(* Logix 5000 project; controller CuteLogix vendor 1 type 14 code 216 rev 30.14; software revision 30.00 *)

TASK EventTask (event, rate 10 ms, priority 10, watchdog 500 ms) : Duh
TASK MainTask (continuous, watchdog 500 ms) : Instructions, Branching

MODULES
   Local : vendor 1 type 14 code 216 (5069 0, rev 30.14)
END_MODULES

TYPE STRING20 :
STRUCT
   LEN : DINT;
   DATA : SINT[20];
END_STRUCT
END_TYPE

VAR_GLOBAL   (* controller tags *)
   AdvancedMath : DINT[10] := ([0] := 651, [3] := 954, [6] := 6);
   ASCII : STRING[20];
   ASCII_Find : DINT;
   ASCII_Find_Result : DINT;
   ASCII_Qty : DINT;
   ASCII_Start : DINT;
   AverageControl : CONTROL := (LEN := 10);
   b_Timer : TIMER[10] := ([0].PRE := 90000, [0].ACC := 52845, [0].EN := 1, [0].TT := 1);
        [0]   // I'm a 90 Second timer
   Bits : DINT[10];
   Branching : DINT[1000] := ([0] := 82407, [1] := 11343, [2] := 76767, [3] := 20431, [4] := 93845, [5] := 88961, [6] := 95802, [7] := 76730, [8] := 78742, [9] := 28858, [10] := 24388, [11] := 98780, [12] := 74194, [13] := 88651, [14] := 97109, [15] := 70489, [16] := 21759, [17] := 12682, [18] := 51608, [19] := 51105, [20] := 34340, [21] := 67477, [22] := 9682, [23] := 52316, [24] := 60079, [25] := 87946, [26] := 25355, [27] := 61705, [28] := 23349, [29] := 32270, [30] := 4523, [31] := 20763, [32] := 39925, [33] := 47227, [34] := 25474, [35] := 90216, [36] := 63189, [37] := 19334, [38] := 13116, [39] := 58964, [40] := 74627, [41] := 92119, [42] := 81781, [43] := 93714, [44] := 35797, [45] := 72290, [46] := 23509, [47] := 2660, [48] := 45984, [49] := 72685, [50] := 48944, [51] := 54255, [52] := 57274, [53] := 86876, [54] := 25860, [55] := 34445, [56] := 55068, [57] := 196, [58] := 23518, [59] := 53104,
        [60] := 75775, [61] := 34032, [62] := 11808, [63] := 83613, [64] := 27078, [65] := 52948, [66] := 91266, [67] := 23342, [68] := 61979, [69] := 88356, [70] := 87538, [71] := 49455, [72] := 73754, [73] := 19956, [74] := 8441, [75] := 44039, [76] := 47792, [77] := 24338, [78] := 1813, [79] := 81080, [80] := 28038, [81] := 22213, [82] := 76032, [83] := 43482, [84] := 43490, [85] := 56586, [86] := 14618, [87] := 67641, [88] := 82887, [89] := 73251, [90] := 36535, [91] := 99267, [92] := 921, [93] := 34224, [94] := 81286, [95] := 89074, [96] := 74192, [97] := 35254, [98] := 70789, [99] := 94903, [100] := 90087, [101] := 75614, [102] := 74924, [103] := 66053, [104] := 67686, [105] := 14094, [106] := 50491, [107] := 19788, [108] := 36949, [109] := 46559, [110] := 33619, [111] := 72776, [112] := 43045, [113] := 66611, [114] := 49748, [115] := 23967, [116] := 66838, [117] := 33653, [118] := 92725, [119] := 32432,
        [120] := 35949, [121] := 75581, [122] := 92310, [123] := 38436, [124] := 62405, [125] := 99027, [126] := 5445, [127] := 23446, [128] := 3634, [129] := 95984, [130] := 50572, [131] := 64179, [132] := 42294, [133] := 43241, [134] := 6544, [135] := 41013, [136] := 98800, [137] := 16177, [138] := 15917, [139] := 31322, [140] := 95598, [141] := 46619, [142] := 76555, [143] := 58340, [144] := 27140, [145] := 10620, [146] := 62592, [147] := 70487, [148] := 12865, [149] := 27943, [150] := 6446, [151] := 12547, [152] := 15055, [153] := 51388, [154] := 85199, [155] := 83609, [156] := 47725, [157] := 55131, [158] := 24907, [159] := 16737, [160] := 43899, [161] := 81924, [162] := 9125, [163] := 64948, [164] := 14057, [165] := 26270, [166] := 26481, [167] := 27516, [168] := 13940, [169] := 41111, [170] := 22715, [171] := 54684, [172] := 27850, [173] := 95551, [174] := 76562, [175] := 10807, [176] := 3604, [177] := 81954, [178] := 85877, [179] := 90731,
        [180] := 50124, [181] := 84444, [182] := 93795, [183] := 58321, [184] := 83942, [185] := 55706, [186] := 21776, [187] := 72127, [188] := 98888, [189] := 98078, [190] := 46603, [191] := 5622, [192] := 2259, [193] := 25464, [194] := 68812, [195] := 39572, [196] := 82910, [197] := 30899, [198] := 41853, [199] := 18720, [200] := 32673, [201] := 51959, [202] := 85552, [203] := 56119, [204] := 37568, [205] := 65908, [206] := 29436, [207] := 79651, [208] := 34700, [209] := 32924, [210] := 83907, [211] := 40689, [212] := 52367, [213] := 8949, [214] := 33429, [215] := 68883, [216] := 57307, [217] := 85633, [218] := 56031, [219] := 3577, [220] := 79663, [221] := 84961, [222] := 38978, [223] := 80380, [224] := 69012, [225] := 39942, [226] := 80323, [227] := 51518, [228] := 32713, [229] := 15043, [230] := 11143, [231] := 84668, [232] := 62808, [233] := 99189, [234] := 72567, [235] := 21806, [236] := 89789, [237] := 79147, [238] := 40667, [239] := 99508,
        [240] := 90600, [241] := 67080, [242] := 66939, [243] := 32495, [244] := 93170, [245] := 53515, [246] := 20470, [247] := 39580, [248] := 483, [249] := 62424, [250] := 1307, [251] := 82788, [252] := 9479, [253] := 67332, [254] := 3775, [255] := 39510, [256] := 4284, [257] := 93272, [258] := 16406, [259] := 65799, [260] := 13395, [261] := 71017, [262] := 52104, [263] := 27877, [264] := 840, [265] := 28148, [266] := 57193, [267] := 76840, [268] := 15114, [269] := 73046, [270] := 48035, [271] := 68111, [272] := 12541, [273] := 80659, [274] := 7877, [275] := 15975, [276] := 56634, [277] := 47037, [278] := 15404, [279] := 7082, [280] := 97238, [281] := 3431, [282] := 79807, [283] := 43357, [284] := 57116, [285] := 78602, [286] := 23732, [287] := 6885, [288] := 94485, [289] := 44571, [290] := 96772, [291] := 35862, [292] := 88252, [293] := 11874, [294] := 63250, [295] := 96749, [296] := 34190, [297] := 12853, [298] := 29560, [299] := 61009,
        [300] := 24219, [301] := 53874, [302] := 98911, [303] := 19166, [304] := 43701, [305] := 69509, [306] := 3825, [307] := 96142, [308] := 42271, [309] := 29331, [310] := 27095, [311] := 39467, [312] := 44548, [313] := 41271, [314] := 87555, [315] := 97136, [316] := 39244, [317] := 16499, [318] := 61732, [319] := 81001, [320] := 81261, [321] := 95891, [322] := 42237, [323] := 43180, [324] := 44778, [325] := 92930, [326] := 54868, [327] := 40795, [328] := 52161, [329] := 19185, [330] := 46809, [331] := 28074, [332] := 11466, [333] := 82810, [334] := 88188, [335] := 72177, [336] := 49604, [337] := 53088, [338] := 16845, [339] := 70569, [340] := 84274, [341] := 92660, [342] := 63169, [343] := 40489, [344] := 26218, [345] := 30561, [346] := 14751, [347] := 75624, [348] := 38033, [349] := 92852, [350] := 85778, [351] := 64491, [352] := 80319, [353] := 8699, [354] := 74387, [355] := 66643, [356] := 62603, [357] := 70896, [358] := 51215, [359] := 45712,
        [360] := 55357, [361] := 77462, [362] := 64150, [363] := 15112, [364] := 85523, [365] := 32571, [366] := 68709, [367] := 30297, [368] := 99879, [369] := 99236, [370] := 14376, [371] := 42664, [372] := 53669, [373] := 22296, [374] := 32196, [375] := 17960, [376] := 42810, [377] := 28932, [378] := 99353, [379] := 54203, [380] := 52001, [381] := 4016, [382] := 41782, [383] := 26979, [384] := 19158, [385] := 41232, [386] := 97013, [387] := 55977, [388] := 62866, [389] := 30951, [390] := 77905, [391] := 86629, [392] := 59774, [393] := 197, [394] := 52381, [395] := 92029, [396] := 94556, [397] := 36193, [398] := 53622, [399] := 26385, [400] := 43506, [401] := 64525, [402] := 50552, [403] := 42062, [404] := 93734, [405] := 66267, [406] := 1973, [407] := 82396, [408] := 20210, [409] := 87, [410] := 31043, [411] := 12651, [412] := 18796, [413] := 74789, [414] := 76255, [415] := 7847, [416] := 88827, [417] := 99325, [418] := 62264, [419] := 83107,
        [420] := 54708, [421] := 81244, [422] := 3333, [423] := 82540, [424] := 76390, [425] := 976, [426] := 94348, [427] := 18663, [428] := 98314, [429] := 90843, [430] := 92080, [431] := 97486, [432] := 42367, [433] := 8830, [434] := 35849, [435] := 15548, [436] := 99329, [437] := 44884, [438] := 60276, [439] := 65875, [440] := 34626, [441] := 31589, [442] := 84178, [443] := 15627, [444] := 14886, [445] := 65838, [446] := 93540, [447] := 14359, [448] := 13136, [449] := 83951, [450] := 94714, [451] := 39093, [452] := 97112, [453] := 22873, [454] := 41442, [455] := 99078, [456] := 11004, [457] := 65685, [458] := 85926, [459] := 55000, [460] := 91532, [461] := 79264, [462] := 3410, [463] := 41917, [464] := 8700, [465] := 15683, [466] := 83367, [467] := 71772, [468] := 14428, [469] := 31148, [470] := 43290, [471] := 73920, [472] := 96383, [473] := 57141, [474] := 28794, [475] := 15145, [476] := 77125, [477] := 35399, [478] := 32019, [479] := 89297,
        [480] := 11057, [481] := 12415, [482] := 54611, [483] := 42077, [484] := 78428, [485] := 33488, [486] := 13887, [487] := 52219, [488] := 37547, [489] := 48567, [490] := 7929, [491] := 45872, [492] := 23879, [493] := 36974, [494] := 97930, [495] := 10005, [496] := 2990, [497] := 51310, [498] := 45690, [499] := 52666, [500] := 16987, [501] := 84869, [502] := 58178, [503] := 95604, [504] := 77205, [505] := 66416, [506] := 46278, [507] := 99665, [508] := 72977, [509] := 58733, [510] := 50420, [511] := 59898, [512] := 18286, [513] := 36589, [514] := 34816, [515] := 47992, [516] := 50582, [517] := 90684, [518] := 46443, [519] := 51027, [520] := 64473, [521] := 72799, [522] := 68183, [523] := 33719, [524] := 81364, [525] := 73595, [526] := 99507, [527] := 47306, [528] := 95179, [529] := 46851, [530] := 86803, [531] := 70881, [532] := 12477, [533] := 75439, [534] := 76539, [535] := 95435, [536] := 45897, [537] := 68412, [538] := 59806, [539] := 8448,
        [540] := 54361, [541] := 83177, [542] := 38861, [543] := 28242, [544] := 24846, [545] := 71585, [546] := 59255, [547] := 99852, [548] := 59975, [549] := 65189, [550] := 78689, [551] := 11674, [552] := 49631, [553] := 89733, [554] := 84628, [555] := 44306, [556] := 69954, [557] := 7239, [558] := 30285, [559] := 49616, [560] := 21695, [561] := 14771, [562] := 902, [563] := 43262, [564] := 32396, [565] := 10532, [566] := 80170, [567] := 22340, [568] := 77422, [569] := 3135, [570] := 24402, [571] := 76735, [572] := 20681, [573] := 94053, [574] := 74442, [575] := 18763, [576] := 9089, [577] := 88936, [578] := 46733, [579] := 47489, [580] := 36126, [581] := 46401, [582] := 56328, [583] := 96948, [584] := 6036, [585] := 61754, [586] := 98282, [587] := 41889, [588] := 9356, [589] := 80694, [590] := 51720, [591] := 56107, [592] := 99379, [593] := 42488, [594] := 63660, [595] := 79873, [596] := 46147, [597] := 44287, [598] := 62154, [599] := 55518,
        [600] := 7753, [601] := 47609, [602] := 31410, [603] := 49961, [604] := 52145, [605] := 16507, [606] := 34414, [607] := 81979, [608] := 23958, [609] := 86010, [610] := 94833, [611] := 89494, [612] := 82851, [613] := 94123, [614] := 60739, [615] := 38788, [616] := 88402, [617] := 62854, [618] := 49018, [619] := 53666, [620] := 9949, [621] := 25600, [622] := 11619, [623] := 73987, [624] := 94764, [625] := 51443, [626] := 42099, [627] := 43731, [628] := 17824, [629] := 20355, [630] := 25854, [631] := 69789, [632] := 6342, [633] := 67396, [634] := 79990, [635] := 20527, [636] := 18543, [637] := 40174, [638] := 10905, [639] := 15107, [640] := 13163, [641] := 12315, [642] := 79884, [643] := 18443, [644] := 64372, [645] := 31725, [646] := 31353, [647] := 31436, [648] := 91466, [649] := 57461, [650] := 73514, [651] := 7803, [652] := 83871, [653] := 95183, [654] := 29573, [655] := 19778, [656] := 58366, [657] := 60531, [658] := 76491, [659] := 47189,
        [660] := 17277, [661] := 81754, [662] := 59413, [663] := 83709, [664] := 10893, [665] := 45396, [666] := 98708, [667] := 59876, [668] := 13826, [669] := 67604, [670] := 55566, [671] := 64210, [672] := 14166, [673] := 41074, [674] := 76431, [675] := 11854, [676] := 63632, [677] := 22463, [678] := 32946, [679] := 49934, [680] := 52913, [681] := 514, [682] := 95943, [683] := 86920, [684] := 80478, [685] := 25993, [686] := 3568, [687] := 53759, [688] := 86334, [689] := 63454, [690] := 54712, [691] := 54196, [692] := 47689, [693] := 75812, [694] := 82587, [695] := 19801, [696] := 38111, [697] := 44003, [698] := 3075, [699] := 37392, [700] := 93416, [701] := 88398, [702] := 33897, [703] := 85847, [704] := 71569, [705] := 6971, [706] := 91687, [707] := 27362, [708] := 55198, [709] := 99697, [710] := 89292, [711] := 25481, [712] := 82481, [713] := 44925, [714] := 19379, [715] := 47317, [716] := 47115, [717] := 14035, [718] := 9678, [719] := 2898,
        [720] := 41216, [721] := 83775, [722] := 44904, [723] := 57107, [724] := 55233, [725] := 44840, [726] := 74361, [727] := 17600, [728] := 18631, [729] := 82287, [730] := 2700, [731] := 60738, [732] := 46652, [733] := 60912, [734] := 51905, [735] := 67154, [736] := 32627, [737] := 15945, [738] := 6478, [739] := 32710, [740] := 44767, [741] := 81659, [742] := 43403, [743] := 16526, [744] := 23636, [745] := 14580, [746] := 60615, [747] := 6854, [748] := 12985, [749] := 20977, [750] := 38155, [751] := 69896, [752] := 78606, [753] := 45117, [754] := 36924, [755] := 81339, [756] := 44488, [757] := 32968, [758] := 69634, [759] := 81380, [760] := 79037, [761] := 55702, [762] := 39094, [763] := 31500, [764] := 57625, [765] := 57132, [766] := 64649, [767] := 84022, [768] := 62957, [769] := 11523, [770] := 65996, [771] := 94131, [772] := 56552, [773] := 23783, [774] := 25433, [775] := 59502, [776] := 64515, [777] := 80652, [778] := 4266, [779] := 68152,
        [780] := 84389, [781] := 24694, [782] := 79259, [783] := 84703, [784] := 80596, [785] := 74624, [786] := 98074, [787] := 3390, [788] := 32057, [789] := 7873, [790] := 20603, [791] := 59444, [792] := 58151, [793] := 75924, [794] := 19190, [795] := 16415, [796] := 47985, [797] := 84559, [798] := 21121, [799] := 38990, [800] := 93540, [801] := 22828, [802] := 59032, [803] := 55447, [804] := 85148, [805] := 17486, [806] := 93438, [807] := 91055, [808] := 75104, [809] := 83127, [810] := 56019, [811] := 67484, [812] := 45150, [813] := 77279, [814] := 86808, [815] := 12229, [816] := 32179, [817] := 23259, [818] := 91876, [819] := 30229, [820] := 89968, [821] := 72891, [822] := 7028, [823] := 43747, [824] := 27889, [825] := 2443, [826] := 89151, [827] := 48814, [828] := 96106, [829] := 63932, [830] := 45306, [831] := 98588, [832] := 97219, [833] := 39477, [834] := 91698, [835] := 90656, [836] := 35504, [837] := 64165, [838] := 52026, [839] := 48456,
        [840] := 72080, [841] := 94201, [842] := 17427, [843] := 67037, [844] := 38528, [845] := 20646, [846] := 37971, [847] := 72563, [848] := 53924, [849] := 35004, [850] := 34397, [851] := 26246, [852] := 63281, [853] := 74035, [854] := 55904, [855] := 96545, [856] := 76341, [857] := 78501, [858] := 86721, [859] := 19100, [860] := 6225, [861] := 41149, [862] := 61826, [863] := 28917, [864] := 83763, [865] := 69988, [866] := 77688, [867] := 83363, [868] := 95651, [869] := 81552, [870] := 486, [871] := 50213, [872] := 44371, [873] := 71109, [874] := 76931, [875] := 75829, [876] := 62668, [877] := 81102, [878] := 80300, [879] := 80686, [880] := 14204, [881] := 28780, [882] := 96869, [883] := 47523, [884] := 36303, [885] := 30274, [886] := 21314, [887] := 61123, [888] := 77651, [889] := 74053, [890] := 62428, [891] := 79484, [892] := 96097, [893] := 41030, [894] := 56604, [895] := 92057, [896] := 92264, [897] := 11036, [898] := 85700, [899] := 18856,
        [900] := 73189, [901] := 26461, [902] := 8888, [903] := 20103, [904] := 95244, [905] := 5577, [906] := 48846, [907] := 4649, [908] := 67044, [909] := 16743, [910] := 50914, [911] := 36861, [912] := 47564, [913] := 46740, [914] := 71045, [915] := 40583, [916] := 72871, [917] := 84923, [918] := 54848, [919] := 81038, [920] := 67903, [921] := 28037, [922] := 18166, [923] := 65853, [924] := 6236, [925] := 74833, [926] := 31786, [927] := 25698, [928] := 1695, [929] := 19536, [930] := 97843, [931] := 33157, [932] := 85756, [933] := 89568, [934] := 41566, [935] := 13093, [936] := 63716, [937] := 28555, [938] := 64458, [939] := 50192, [940] := 68170, [941] := 94118, [942] := 6870, [943] := 15809, [944] := 41960, [945] := 90340, [946] := 89635, [947] := 25943, [948] := 46729, [949] := 96818, [950] := 59347, [951] := 16070, [952] := 37787, [953] := 1937, [954] := 20945, [955] := 63579, [956] := 67266, [957] := 14286, [958] := 85165, [959] := 43977,
        [960] := 58184, [961] := 2173, [962] := 53896, [963] := 1423, [964] := 45727, [965] := 35643, [966] := 77499, [967] := 66850, [968] := 26190, [969] := 36629, [970] := 60325, [971] := 1963, [972] := 25057, [973] := 56880, [974] := 44853, [975] := 91039, [976] := 40727, [977] := 70695, [978] := 49373, [979] := 15523, [980] := 55032, [981] := 51073, [982] := 7087, [983] := 49070, [984] := 87957, [985] := 10121, [986] := 89376, [987] := 92311, [988] := 40916, [989] := 78216, [990] := 33126, [991] := 90167, [992] := 14188, [993] := 10078, [994] := 66544, [995] := 16155, [996] := 50291, [997] := 33595, [998] := 17181, [999] := 38750);
   BSLControl : CONTROL := (LEN := 10);
   BSRControl : CONTROL := (LEN := 66);
   CmpControl : CONTROL := (LEN := 10);
   Controller_Name : STRING;
   Conv_BCD : DINT[10] := ([1] := 22);
   Counters : COUNTER[5] := ([0].PRE := 984684);
   Dint_Conv : DINT[10] := ([0] := 88);
   DisableWeb : SINT[5] := ([0] := 1, [1] := 80, [3] := 6);
   EOT_Test : BOOL;
   FAL_Dest : DINT := 88;
   FALControl : CONTROL := (LEN := 10);
   False : BOOL := 1;
   FaultCounter : COUNTER := (PRE := 2147483647, ACC := 1584);   // I count stuff
   FFLControl : CONTROL := (LEN := 48, POS := 4);
   FFU_Dest : DINT;
   FirstOutFault : DINT;
   For_Index : DINT;
   FSCControl : CONTROL := (LEN := 10, POS := 4);
   Immediate_Out : DINT;
   LFLControl : CONTROL := (LEN := 10, POS := 6);
   LFU_Dest : DINT;
   Logicals : DINT[20] := ([0] := 53762, [1] := 42738, [2] := 55791, [3] := 6185, [4] := 59046, [5] := 47924, [6] := 57863, [7] := 44456, [8] := 54033, [9] := 34837, [10] := 4227, [11] := 32054, [12] := 427, [13] := 63322, [14] := 8111, [15] := 29684, [16] := 22372, [17] := 36781, [18] := 42828, [19] := 58861);
   m_MAFR : MOTION_INSTRUCTION;
   m_MAS : MOTION_INSTRUCTION;
   m_MASD : MOTION_INSTRUCTION;
   m_MASR : MOTION_INSTRUCTION;
   MathConv : REAL[20] := ([1] := 6.0);
   Maths : DINT[20] := ([0] := 13510, [1] := 32560, [2] := 48848, [3] := 20552, [4] := 54861, [5] := 701, [6] := 10281, [7] := 25882, [8] := 16938, [9] := 48231, [10] := 47695, [11] := 37374, [12] := 55424, [13] := 20245, [14] := 51775, [15] := 55217, [16] := 43048, [17] := 38304, [18] := 47601, [19] := 2516);
   Maths_Dest : DINT := 666;
   Message : MESSAGE;
   Misc : DINT[10];
   Misc_Average : DINT;
   Misc_IO : DINT;
   Misc_Size : DINT;
   Misc_STD : REAL;
   MiscArray : DINT[10];
   PID_CV : DINT;
   PID_Inhold : BOOL;
   PID_Inhold_Value : DINT;
   PID_Master : PID;
   PID_PV : DINT;
   PID_Tieback : DINT;
   Real_Conf : REAL[10];
   ResControl : CONTROL := (LEN := 10);
   Ret_Parameter : DINT;
   SBR_Parameter : DINT;
   SeqArray : DINT[10];
   SeqControl : CONTROL := (LEN := 10);
   SeqDest : DINT;
   SeqMask : DINT;
   SeqSource : DINT;
   ShiftArray : DINT[20];
   ShiftBits : DINT;
   ShiftFIFO : DINT[10];
   ShiftLFL : DINT[10];
   SortControl : CONTROL := (LEN := 10, POS := 8);
   Special : DINT[20];
   Special_PID : PID := (SP := 50.0);
   STDControl : CONTROL := (LEN := 10);
   Str_Conv : STRING[10] := ([0] := '10', [2] := '42.0');
   Task_State : DINT;
   ThatTag : DINT;
   ThisMask : DINT := 456789;
   ThisTag : DINT := 99;   // Stuff
   Timers : TIMER[5] := ([0].PRE := 1000, [0].ACC := 123, [1].PRE := 1364686, [1].ACC := 456, [2].PRE := 5500, [2].ACC := 456);
   Toggle : BOOL;
   Trig : REAL[20] := ([0] := 16.45, [1] := 6.66, [2] := 18.1, [3] := 42.0, [4] := 2.0, [8] := 0.45);
   VAxis : AXIS_VIRTUAL;
   WebPage : MESSAGE;
        MessageParameters(ServiceCode := 16#004c, LocalElement := DisableWeb[0], ...)
   WhyIsThisNecessary : MOTION_GROUP;
END_VAR

PROGRAM Branching   (* main routine B001_Main *)

ROUTINE B001_Main   (* ladder *)
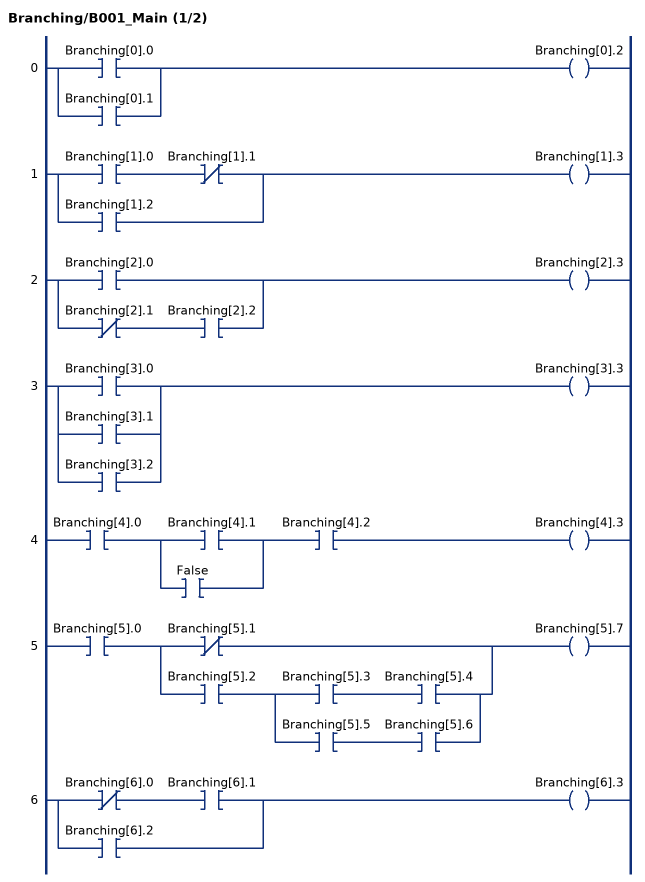
   0: [XIC(Branching[0].0) ,XIC(Branching[0].1) ]OTE(Branching[0].2);
   1: [XIC(Branching[1].0) XIO(Branching[1].1) ,XIC(Branching[1].2) ]OTE(Branching[1].3);
   2: [XIC(Branching[2].0) ,XIO(Branching[2].1) XIC(Branching[2].2) ]OTE(Branching[2].3);
   3: [XIC(Branching[3].0) ,XIC(Branching[3].1) ,XIC(Branching[3].2) ]OTE(Branching[3].3);
   4: XIC(Branching[4].0)[XIC(Branching[4].1) ,XIC(False) ]XIC(Branching[4].2)OTE(Branching[4].3);
   5: XIC(Branching[5].0)[XIO(Branching[5].1) ,XIC(Branching[5].2) [XIC(Branching[5].3) XIC(Branching[5].4) ,XIC(Branching[5].5) XIC(Branching[5].6) ] ]OTE(Branching[5].7);
   6: [XIO(Branching[6].0) XIC(Branching[6].1) ,XIC(Branching[6].2) ]OTE(Branching[6].3);
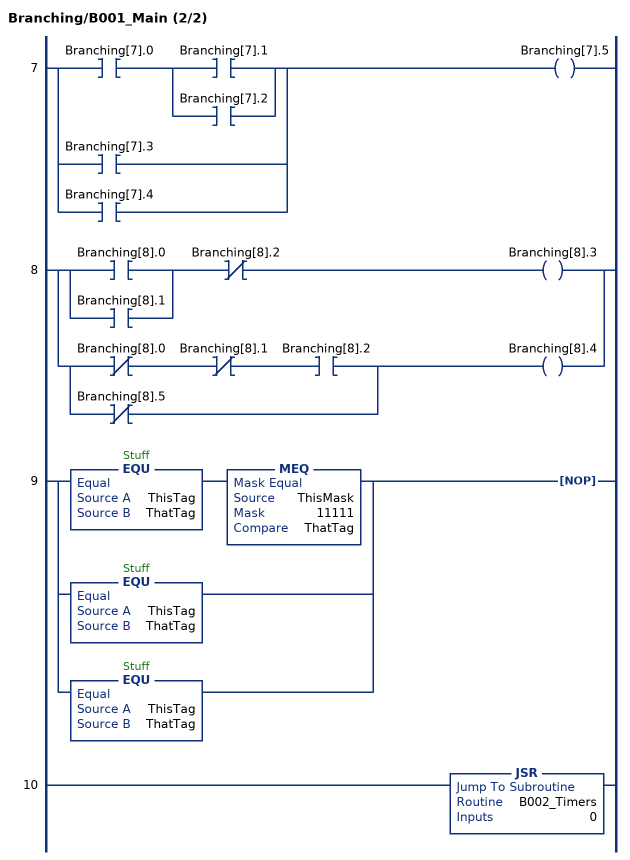
   7: [XIC(Branching[7].0) [XIC(Branching[7].1) ,XIC(Branching[7].2) ] ,XIC(Branching[7].3) ,XIC(Branching[7].4) ]OTE(Branching[7].5);
   8: [[XIC(Branching[8].0) ,XIC(Branching[8].1) ] XIO(Branching[8].2) OTE(Branching[8].3) ,[XIO(Branching[8].0) XIO(Branching[8].1) XIC(Branching[8].2) ,XIO(Branching[8].5) ] OTE(Branching[8].4) ];
   9: [EQU(ThisTag,ThatTag) MEQ(ThisMask,11111,ThatTag) ,EQU(ThisTag,ThatTag) ,EQU(ThisTag,ThatTag) ]NOP();
   10: JSR(B002_Timers,0);
END_ROUTINE

ROUTINE B002_Timers   (* ladder *)
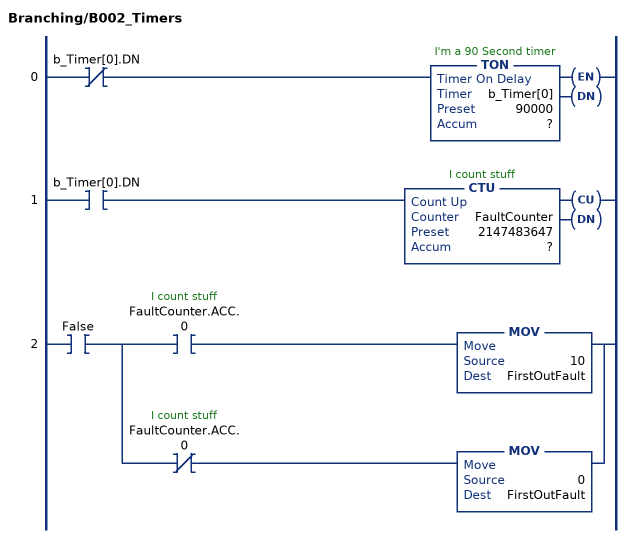
   0: XIO(b_Timer[0].DN)TON(b_Timer[0],?,?);
   1: XIC(b_Timer[0].DN)CTU(FaultCounter,?,?);
   2: XIC(False)[XIC(FaultCounter.ACC.0) MOV(10,FirstOutFault) ,XIO(FaultCounter.ACC.0) MOV(0,FirstOutFault) ];
END_ROUTINE
END_PROGRAM

PROGRAM Duh   (* main routine Stupid *)

ROUTINE Stupid   (* ladder *)
   0: NOP();
END_ROUTINE
END_PROGRAM

PROGRAM Instructions   (* main routine MainRoutine *)

ROUTINE MainRoutine   (* ladder *)
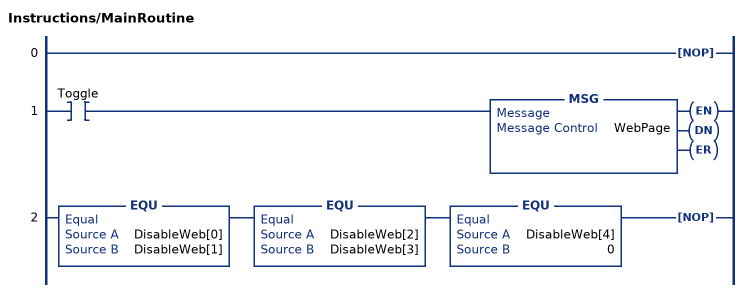
   0: NOP();
   1: XIC(Toggle)MSG(WebPage);
   2: EQU(DisableWeb[0],DisableWeb[1])EQU(DisableWeb[2],DisableWeb[3])EQU(DisableWeb[4],0)NOP();
END_ROUTINE

ROUTINE R010_Bit   (* ladder *)
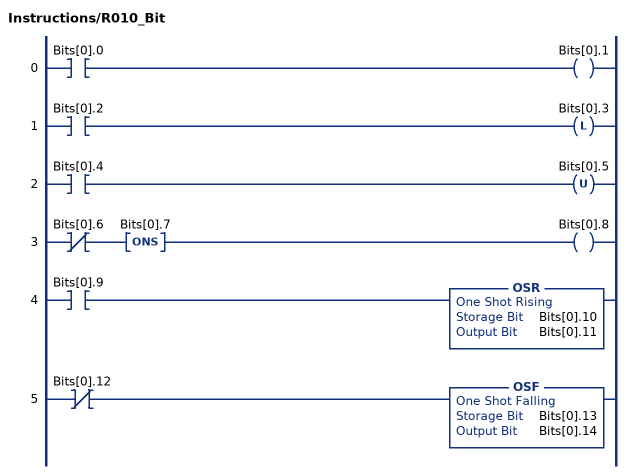
   0: XIC(Bits[0].0)OTE(Bits[0].1);
   1: XIC(Bits[0].2)OTL(Bits[0].3);
   2: XIC(Bits[0].4)OTU(Bits[0].5);
   3: XIO(Bits[0].6)ONS(Bits[0].7)OTE(Bits[0].8);
   4: XIC(Bits[0].9)OSR(Bits[0].10,Bits[0].11);
   5: XIO(Bits[0].12)OSF(Bits[0].13,Bits[0].14);
END_ROUTINE

ROUTINE R011_Timer_Counter   (* ladder *)
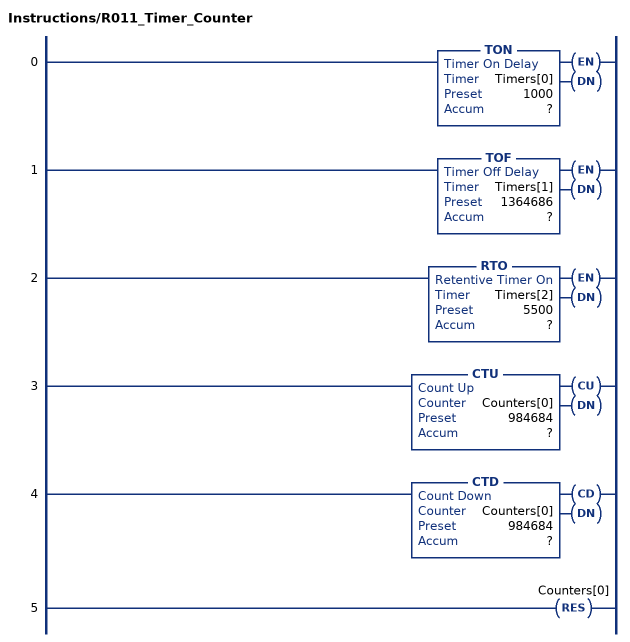
   0: TON(Timers[0],?,?);
   1: TOF(Timers[1],?,?);
   2: RTO(Timers[2],?,?);
   3: CTU(Counters[0],?,?);
   4: CTD(Counters[0],?,?);
   5: RES(Counters[0]);
END_ROUTINE

ROUTINE R012_Input_Output   (* ladder *)
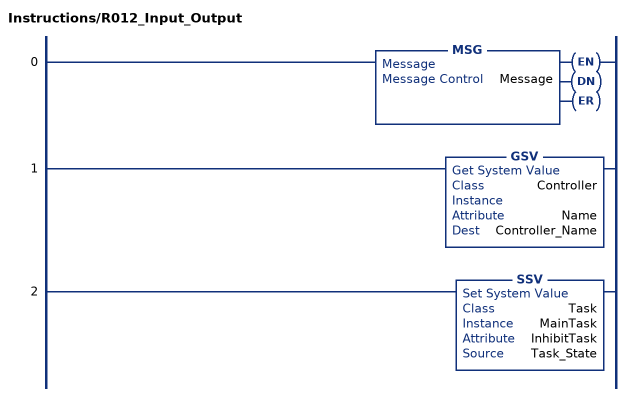
   0: MSG(Message);
   1: GSV(Controller,,Name,Controller_Name);
   2: SSV(Task,MainTask,InhibitTask,Task_State);
END_ROUTINE

ROUTINE R013_Compare   (* ladder *)
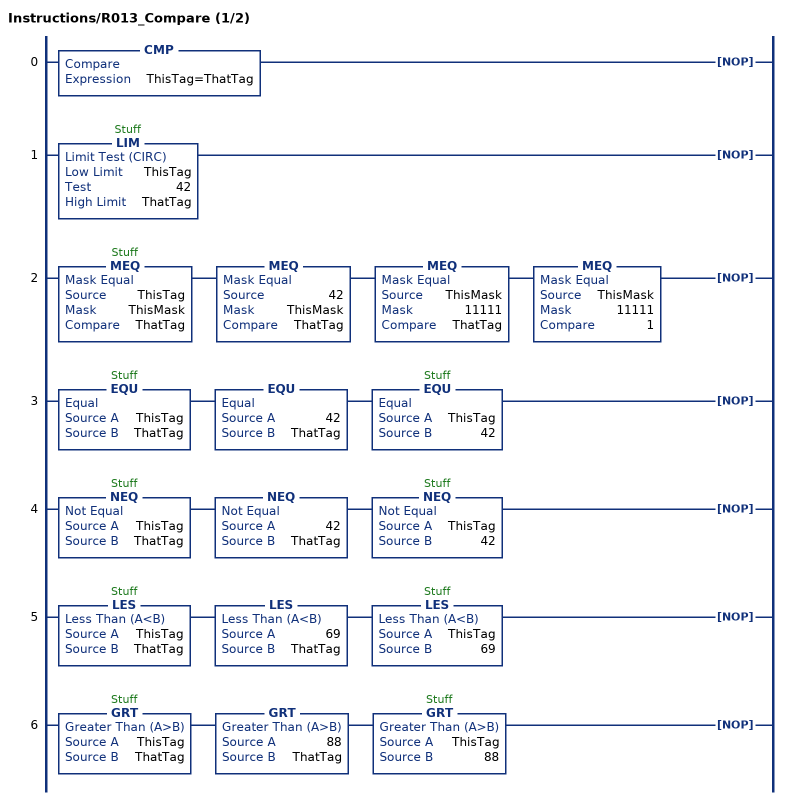
   0: CMP(ThisTag=ThatTag)NOP();
   1: LIM(ThisTag,42,ThatTag)NOP();
   2: MEQ(ThisTag,ThisMask,ThatTag)MEQ(42,ThisMask,ThatTag)MEQ(ThisMask,11111,ThatTag)MEQ(ThisMask,11111,1)NOP();
   3: EQU(ThisTag,ThatTag)EQU(42,ThatTag)EQU(ThisTag,42)NOP();
   4: NEQ(ThisTag,ThatTag)NEQ(42,ThatTag)NEQ(ThisTag,42)NOP();
   5: LES(ThisTag,ThatTag)LES(69,ThatTag)LES(ThisTag,69)NOP();
   6: GRT(ThisTag,ThatTag)GRT(88,ThatTag)GRT(ThisTag,88)NOP();
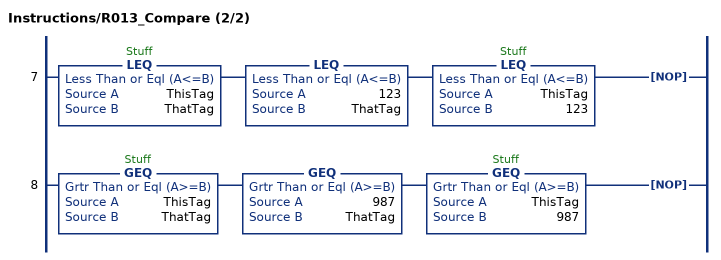
   7: LEQ(ThisTag,ThatTag)LEQ(123,ThatTag)LEQ(ThisTag,123)NOP();
   8: GEQ(ThisTag,ThatTag)GEQ(987,ThatTag)GEQ(ThisTag,987)NOP();
END_ROUTINE

ROUTINE R014_Compute_Math   (* ladder *)
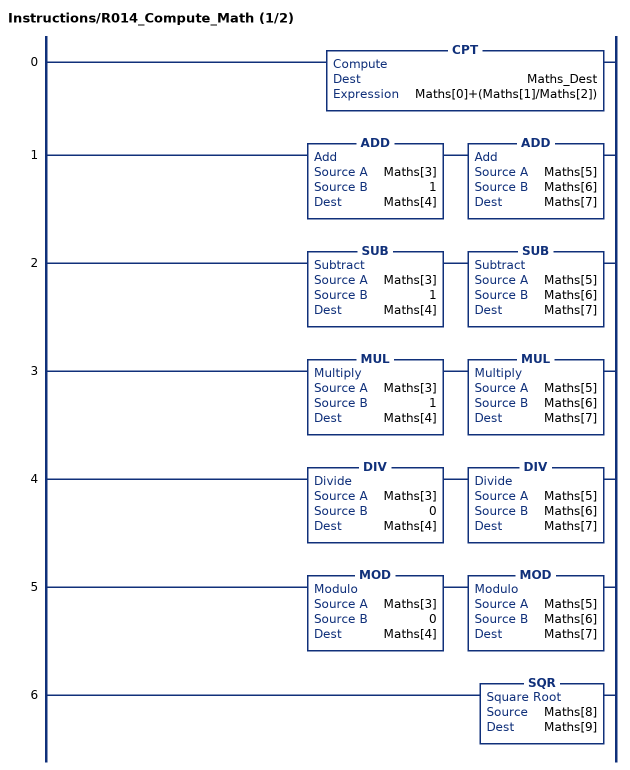
   0: CPT(Maths_Dest,Maths[0]+(Maths[1]/Maths[2]));
   1: ADD(Maths[3],1,Maths[4])ADD(Maths[5],Maths[6],Maths[7]);
   2: SUB(Maths[3],1,Maths[4])SUB(Maths[5],Maths[6],Maths[7]);
   3: MUL(Maths[3],1,Maths[4])MUL(Maths[5],Maths[6],Maths[7]);
   4: DIV(Maths[3],0,Maths[4])DIV(Maths[5],Maths[6],Maths[7]);
   5: MOD(Maths[3],0,Maths[4])MOD(Maths[5],Maths[6],Maths[7]);
   6: SQR(Maths[8],Maths[9]);
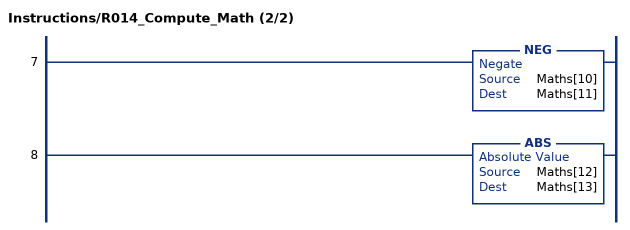
   7: NEG(Maths[10],Maths[11]);
   8: ABS(Maths[12],Maths[13]);
END_ROUTINE

ROUTINE R015_Move_Logical   (* ladder *)
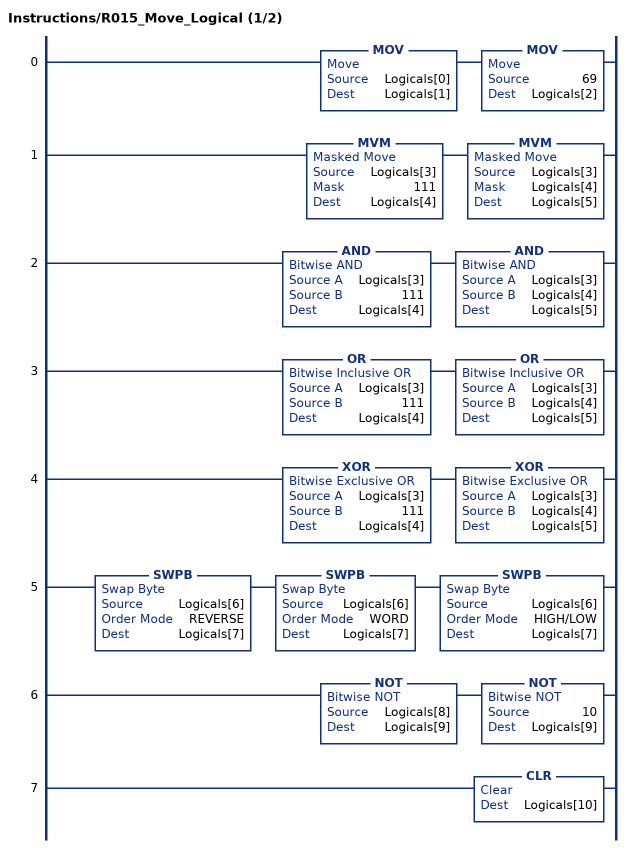
   0: MOV(Logicals[0],Logicals[1])MOV(69,Logicals[2]);
   1: MVM(Logicals[3],111,Logicals[4])MVM(Logicals[3],Logicals[4],Logicals[5]);
   2: AND(Logicals[3],111,Logicals[4])AND(Logicals[3],Logicals[4],Logicals[5]);
   3: OR(Logicals[3],111,Logicals[4])OR(Logicals[3],Logicals[4],Logicals[5]);
   4: XOR(Logicals[3],111,Logicals[4])XOR(Logicals[3],Logicals[4],Logicals[5]);
   5: SWPB(Logicals[6],REVERSE,Logicals[7])SWPB(Logicals[6],WORD,Logicals[7])SWPB(Logicals[6],HIGH/LOW,Logicals[7]);
   6: NOT(Logicals[8],Logicals[9])NOT(10,Logicals[9]);
   7: CLR(Logicals[10]);
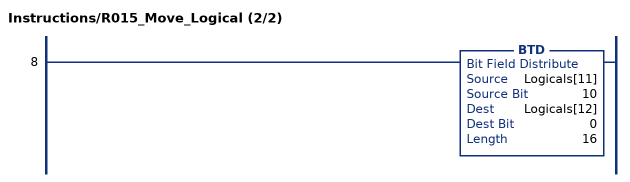
   8: BTD(Logicals[11],10,Logicals[12],0,16);
END_ROUTINE

ROUTINE R016_File_Misc   (* ladder *)
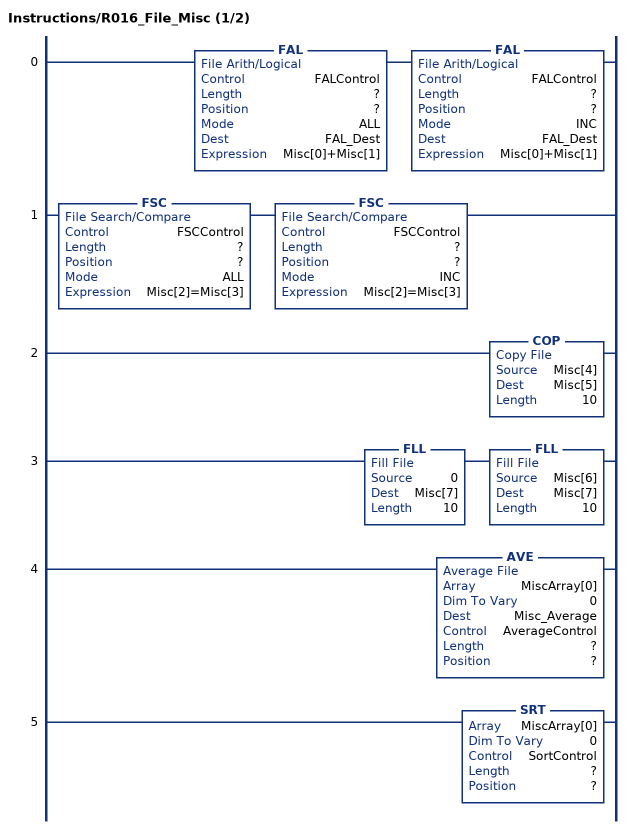
   0: FAL(FALControl,?,?,ALL,FAL_Dest,Misc[0]+Misc[1])FAL(FALControl,?,?,INC,FAL_Dest,Misc[0]+Misc[1]);
   1: FSC(FSCControl,?,?,ALL,Misc[2]=Misc[3])FSC(FSCControl,?,?,INC,Misc[2]=Misc[3]);
   2: COP(Misc[4],Misc[5],10);
   3: FLL(0,Misc[7],10)FLL(Misc[6],Misc[7],10);
   4: AVE(MiscArray[0],0,Misc_Average,AverageControl,?,?);
   5: SRT(MiscArray[0],0,SortControl,?,?);
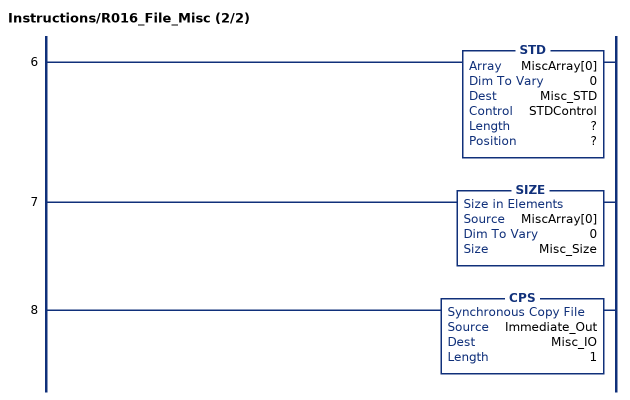
   6: STD(MiscArray[0],0,Misc_STD,STDControl,?,?);
   7: SIZE(MiscArray[0],0,Misc_Size);
   8: CPS(Immediate_Out,Misc_IO,1);
END_ROUTINE

ROUTINE R017_File_Shift   (* ladder *)
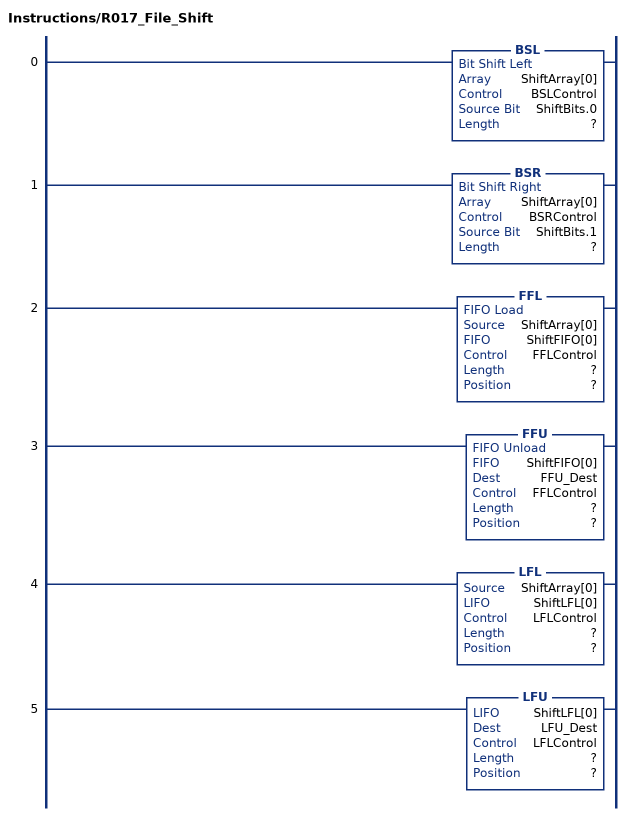
   0: BSL(ShiftArray[0],BSLControl,ShiftBits.0,?);
   1: BSR(ShiftArray[0],BSRControl,ShiftBits.1,?);
   2: FFL(ShiftArray[0],ShiftFIFO[0],FFLControl,?,?);
   3: FFU(ShiftFIFO[0],FFU_Dest,FFLControl,?,?);
   4: LFL(ShiftArray[0],ShiftLFL[0],LFLControl,?,?);
   5: LFU(ShiftLFL[0],LFU_Dest,LFLControl,?,?);
END_ROUTINE

ROUTINE R018_Sequencer   (* ladder *)
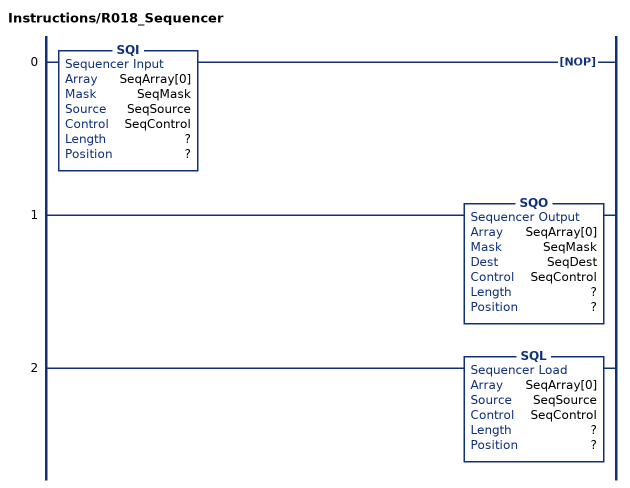
   0: SQI(SeqArray[0],SeqMask,SeqSource,SeqControl,?,?)NOP();
   1: SQO(SeqArray[0],SeqMask,SeqDest,SeqControl,?,?);
   2: SQL(SeqArray[0],SeqSource,SeqControl,?,?);
END_ROUTINE

ROUTINE R019_Equipment_Phase   (* ladder *)
   0: NOP();
END_ROUTINE

ROUTINE R020_Program_Control   (* ladder *)
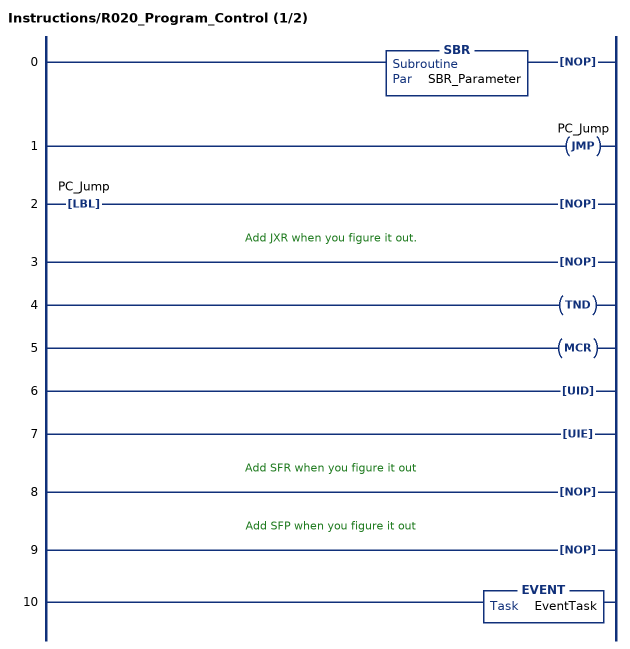
   0: SBR(SBR_Parameter)NOP();
   1: JMP(PC_Jump);
   2: LBL(PC_Jump)NOP();
   // Add JXR when you figure it out.
   3: NOP();
   4: TND();
   5: MCR();
   6: UID();
   7: UIE();
   // Add SFR when you figure it out
   8: NOP();
   // Add SFP when you figure it out
   9: NOP();
   10: EVENT(EventTask);
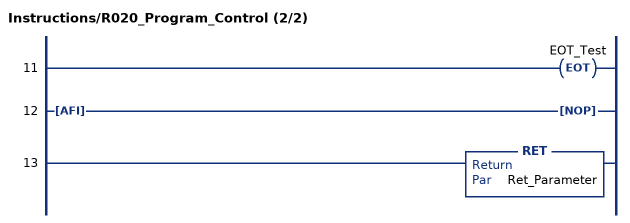
   11: EOT(EOT_Test);
   12: AFI()NOP();
   13: RET(Ret_Parameter);
END_ROUTINE
